// Mitsubishi GX Works2 project: conorGleesonAssignment   PLC: FX2N/FX2NC

PROGRAM MAIN
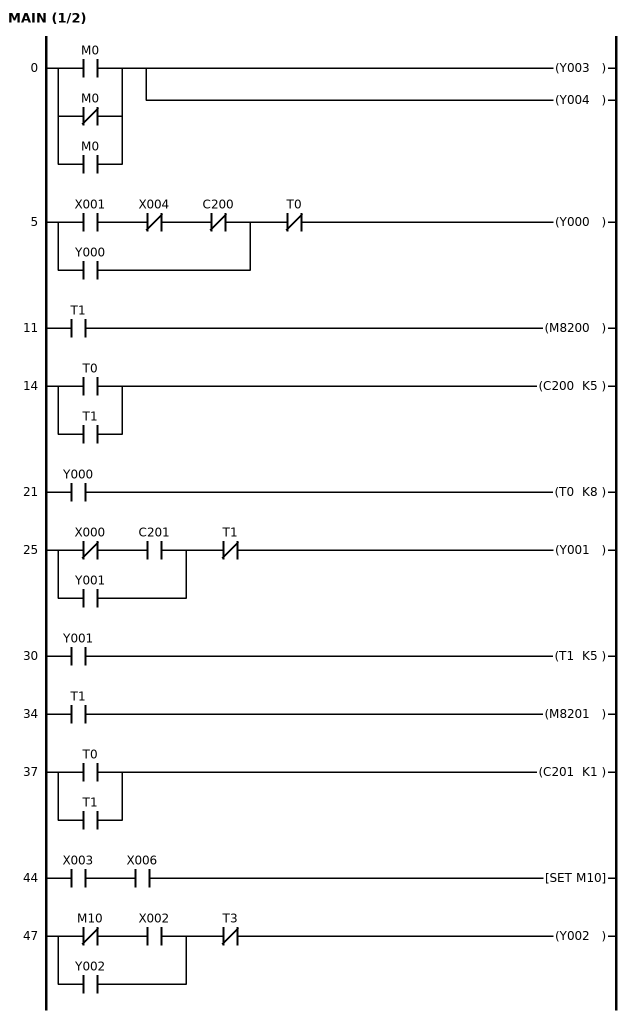
0     LD      M0
      ORI     M0
      OR      M0
      OUT     Y003
      OUT     Y004
5     LD      X001
      ANI     X004
      ANI     C200
      OR      Y000
      ANI     T0
      OUT     Y000
11    LD      T1
      OUT     M8200
14    LD      T0
      OR      T1
      OUT     C200 K5
21    LD      Y000
      OUT     T0 K8
25    LDI     X000
      AND     C201
      OR      Y001
      ANI     T1
      OUT     Y001
30    LD      Y001
      OUT     T1 K5
34    LD      T1
      OUT     M8201
37    LD      T0
      OR      T1
      OUT     C201 K1
44    LD      X003
      AND     X006
      SET     M10
47    LDI     M10
      AND     X002
      OR      Y002
      ANI     T3
      OUT     Y002
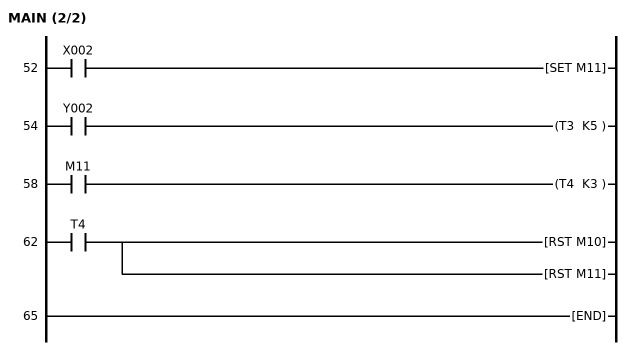
52    LD      X002
      SET     M11
54    LD      Y002
      OUT     T3 K5
58    LD      M11
      OUT     T4 K3
62    LD      T4
      RST     M10
      RST     M11
65    END
END_PROGRAM
